// Mitsubishi GX Works2 project: SET_RESET   PLC: Q03UDV

PROGRAM MAIN
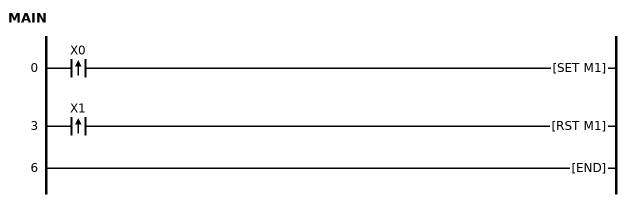
0     LDP     X0
      SET     M1
3     LDP     X1
      RST     M1
6     END
END_PROGRAM
